FUNCTION_BLOCK fb_Blink
VAR_INPUT
	tLowTime		: TIME;
	tCycleTime	: TIME;
END_VAR
VAR_OUTPUT
	bCycle			: BOOL;
END_VAR
VAR
	tonLowTime		: TON;
	tofCycleTime	: TOF;
END_VAR

tonLowTime(IN:=(NOT tofCycleTime.Q), PT:= tLowTime);
tofCycleTime(IN:=(tonLowTime.Q), PT:= tCycleTime);

bCycle := tofCycleTime.Q;

END_FUNCTION_BLOCK

(* stored: Version 1.1.0.1, ProductVersion 3.1.4024.9
   POU fb_Blink: Id {62267eda-500d-4f86-91b2-9237e804b825}, SpecialFunc None *)
